// TIA Portal V17 export
// export: Created 2024-08-26T21:07:16.8648611Z, ExportSetting WithDefaults, DisplayName Totally Integrated Automation Portal, DisplayVersion V17 Update 7, DisplayName TIA Portal Openness, DisplayVersion V17 Update 7, DisplayName TIA Portal Version Control Interface, DisplayVersion V17, DisplayName SINAMICS Startdrive Advanced, DisplayVersion V17 SP2, DisplayName SINAMICS Startdrive G110M, G120, G120C, G120D, G120P, G115D, DisplayVersion V17 SP2, DisplayName SINAMICS Startdrive G130, G150, S120, S150, SINAMICS MV, S210, DisplayVersion V17 SP2, DisplayName STEP 7 Professional, DisplayVersion V17 Update 7, DisplayName STEP 7 Safety, DisplayVersion V17 Update 6, DisplayName WinCC Advanced / Unified PC, DisplayVersion V17 Update 7
FUNCTION "SCANNER CONFIG" : Void   // FC11, LAD
{ S7_Optimized_Access := 'TRUE' }
VERSION : 0.1
// stored: AutoNumber true, IsIECCheckEnabled false, SetENOAutomatically false, UDAEnableTagReadback false
   VAR_TEMP   // added for the SCL form of the ladder/FBD networks
      _w1 : Bool;
   END_VAR
BEGIN

REGION Network 1: NEST CODE READING
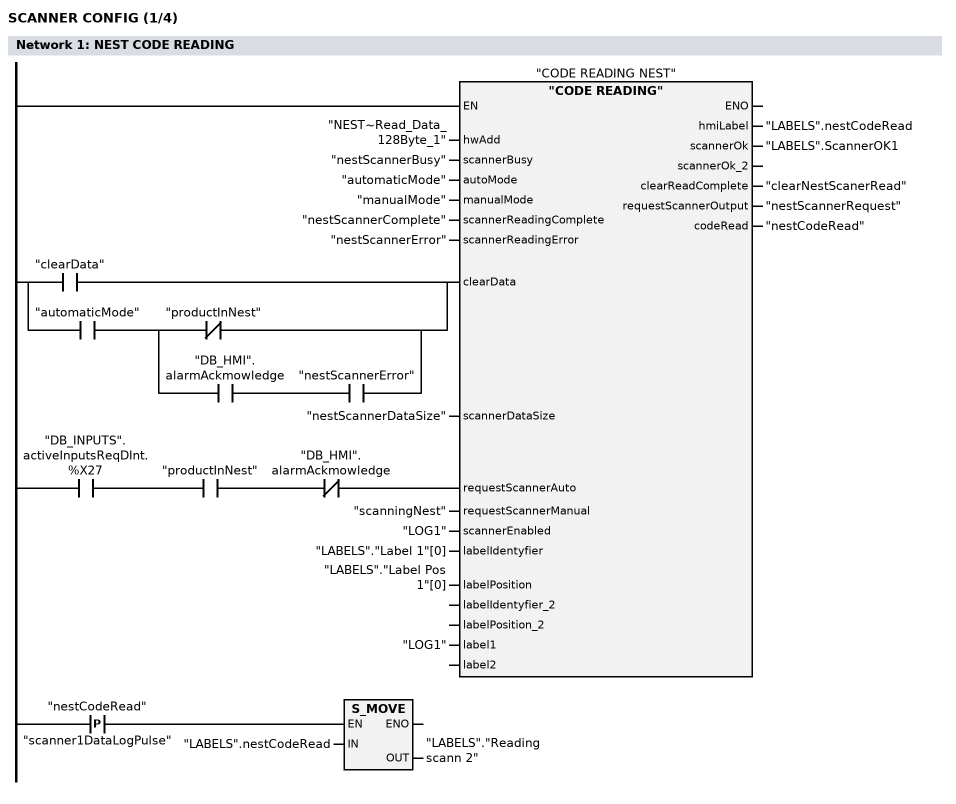
   RUNG wire#powerrail
      "CODE READING NEST"(clearData := wire#w2, requestScannerAuto := wire#w3, hwAdd := "NEST~Read_Data_128Byte_1", scannerBusy := "nestScannerBusy", autoMode := "automaticMode", manualMode := "manualMode", scannerReadingComplete := "nestScannerComplete", scannerReadingError := "nestScannerError", scannerDataSize := "nestScannerDataSize", requestScannerManual := "scanningNest", scannerEnabled := "LOG1", labelIdentyfier := "LABELS"."Label 1"[0], labelPosition := "LABELS"."Label Pos 1"[0], labelIdentyfier_2 :=, labelPosition_2 :=, label1 := "LOG1", label2 :=, hmiLabel => "LABELS".nestCodeRead, scannerOk => "LABELS".ScannerOK1, scannerOk_2 =>, clearReadComplete => "clearNestScanerRead", requestScannerOutput => "nestScannerRequest", codeRead => "nestCodeRead")
   END_RUNG
   RUNG wire#powerrail
      Contact( "clearData" )
   END_RUNG wire#w2
   RUNG wire#powerrail
      Contact( "automaticMode" )
      wire#w1
      I_Contact( "productInNest" )
   END_RUNG wire#w2
   RUNG wire#w1
      Contact( "DB_HMI".alarmAckmowledge )
      Contact( "nestScannerError" )
   END_RUNG wire#w2
   RUNG wire#powerrail
      Contact( "DB_INPUTS".activeInputsReqDInt.%X27 )
      Contact( "productInNest" )
      I_Contact( "DB_HMI".alarmAckmowledge )
   END_RUNG wire#w3
   RUNG wire#powerrail
      P_Contact(operand := "nestCodeRead", bit := "scanner1DataLogPulse")
      S_Move(in := "LABELS".nestCodeRead, out => "LABELS"."Reading scann 2")
   END_RUNG
   // the same network as SCL:
   "CODE READING NEST"(hwAdd := "NEST~Read_Data_128Byte_1",   // "CODE READING"
                       scannerBusy := "nestScannerBusy",
                       autoMode := "automaticMode",
                       manualMode := "manualMode",
                       scannerReadingComplete := "nestScannerComplete",
                       scannerReadingError := "nestScannerError",
                       clearData := "clearData" OR ("automaticMode" AND (NOT "productInNest" OR ("DB_HMI".alarmAckmowledge AND "nestScannerError"))),
                       scannerDataSize := "nestScannerDataSize",
                       requestScannerAuto := "DB_INPUTS".activeInputsReqDInt.%X27 AND "productInNest" AND NOT "DB_HMI".alarmAckmowledge,
                       requestScannerManual := "scanningNest",
                       scannerEnabled := "LOG1",
                       labelIdentyfier := "LABELS"."Label 1"[0],
                       labelPosition := "LABELS"."Label Pos 1"[0],
                       label1 := "LOG1",
                       hmiLabel => "LABELS".nestCodeRead,
                       scannerOk => "LABELS".ScannerOK1,
                       clearReadComplete => "clearNestScanerRead",
                       requestScannerOutput => "nestScannerRequest",
                       codeRead => "nestCodeRead");
   #_w1 := "nestCodeRead" AND NOT "scanner1DataLogPulse";   // rising edge of "nestCodeRead"
   "scanner1DataLogPulse" := "nestCodeRead";
   IF #_w1 THEN "LABELS"."Reading scann 2" := "LABELS".nestCodeRead; END_IF;
END_REGION

REGION Network 2: UPPER CODE READING
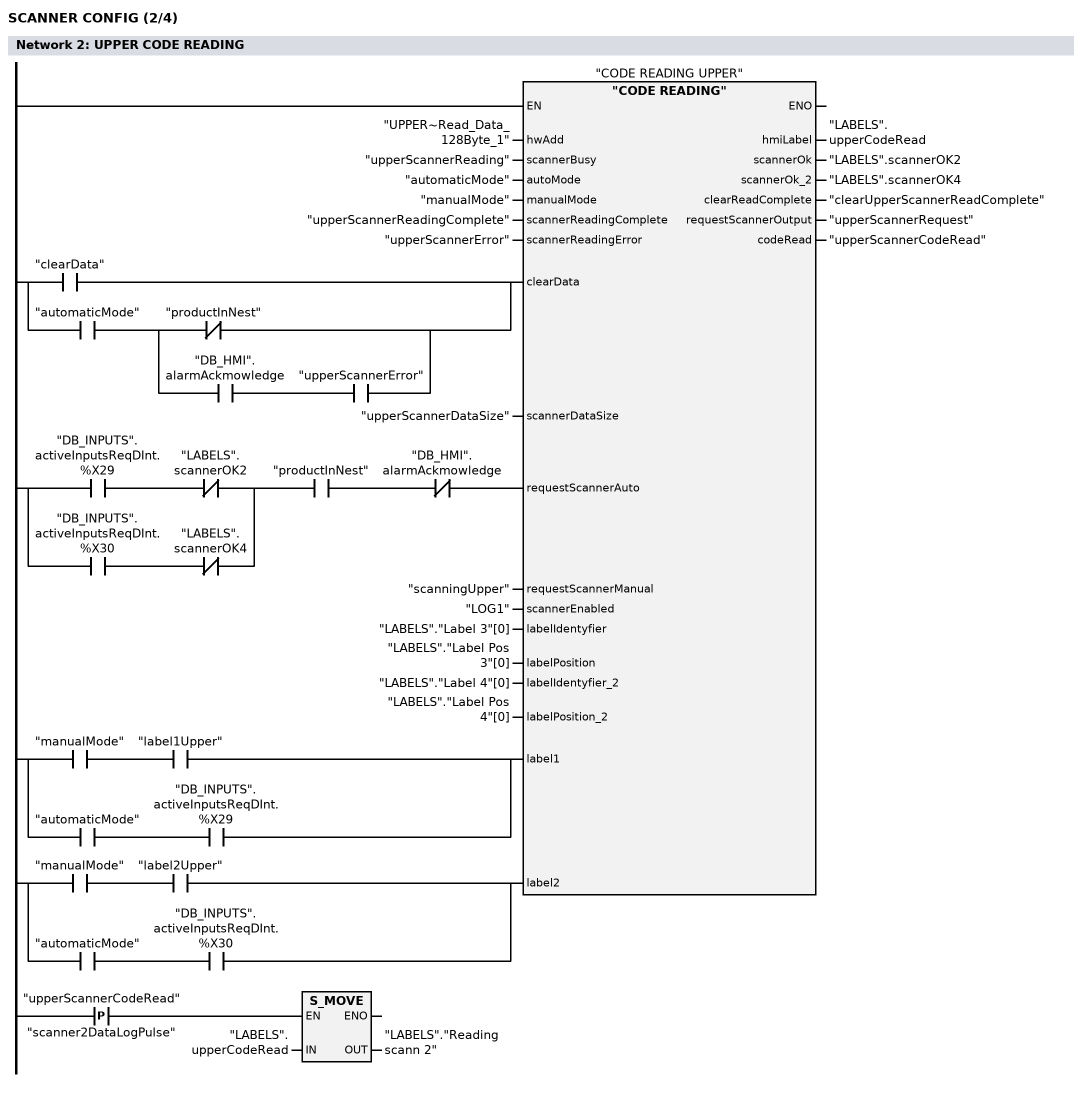
   RUNG wire#powerrail
      "CODE READING UPPER"(clearData := wire#w2, requestScannerAuto := wire#w4, label1 := wire#w5, label2 := wire#w6, hwAdd := "UPPER~Read_Data_128Byte_1", scannerBusy := "upperScannerReading", autoMode := "automaticMode", manualMode := "manualMode", scannerReadingComplete := "upperScannerReadingComplete", scannerReadingError := "upperScannerError", scannerDataSize := "upperScannerDataSize", requestScannerManual := "scanningUpper", scannerEnabled := "LOG1", labelIdentyfier := "LABELS"."Label 3"[0], labelPosition := "LABELS"."Label Pos 3"[0], labelIdentyfier_2 := "LABELS"."Label 4"[0], labelPosition_2 := "LABELS"."Label Pos 4"[0], hmiLabel => "LABELS".upperCodeRead, scannerOk => "LABELS".scannerOK2, scannerOk_2 => "LABELS".scannerOK4, clearReadComplete => "clearUpperScannerReadComplete", requestScannerOutput => "upperScannerRequest", codeRead => "upperScannerCodeRead")
   END_RUNG
   RUNG wire#powerrail
      Contact( "clearData" )
   END_RUNG wire#w2
   RUNG wire#powerrail
      Contact( "automaticMode" )
      wire#w1
      I_Contact( "productInNest" )
   END_RUNG wire#w2
   RUNG wire#w1
      Contact( "DB_HMI".alarmAckmowledge )
      Contact( "upperScannerError" )
   END_RUNG wire#w2
   RUNG wire#powerrail
      Contact( "DB_INPUTS".activeInputsReqDInt.%X29 )
      I_Contact( "LABELS".scannerOK2 )
      wire#w3
      Contact( "productInNest" )
      I_Contact( "DB_HMI".alarmAckmowledge )
   END_RUNG wire#w4
   RUNG wire#powerrail
      Contact( "DB_INPUTS".activeInputsReqDInt.%X30 )
      I_Contact( "LABELS".scannerOK4 )
   END_RUNG wire#w3
   RUNG wire#powerrail
      Contact( "manualMode" )
      Contact( "label1Upper" )
   END_RUNG wire#w5
   RUNG wire#powerrail
      Contact( "automaticMode" )
      Contact( "DB_INPUTS".activeInputsReqDInt.%X29 )
   END_RUNG wire#w5
   RUNG wire#powerrail
      Contact( "manualMode" )
      Contact( "label2Upper" )
   END_RUNG wire#w6
   RUNG wire#powerrail
      Contact( "automaticMode" )
      Contact( "DB_INPUTS".activeInputsReqDInt.%X30 )
   END_RUNG wire#w6
   RUNG wire#powerrail
      P_Contact(operand := "upperScannerCodeRead", bit := "scanner2DataLogPulse")
      S_Move(in := "LABELS".upperCodeRead, out => "LABELS"."Reading scann 2")
   END_RUNG
   // the same network as SCL:
   "CODE READING UPPER"(hwAdd := "UPPER~Read_Data_128Byte_1",   // "CODE READING"
                        scannerBusy := "upperScannerReading",
                        autoMode := "automaticMode",
                        manualMode := "manualMode",
                        scannerReadingComplete := "upperScannerReadingComplete",
                        scannerReadingError := "upperScannerError",
                        clearData := "clearData" OR ("automaticMode" AND (NOT "productInNest" OR ("DB_HMI".alarmAckmowledge AND "upperScannerError"))),
                        scannerDataSize := "upperScannerDataSize",
                        requestScannerAuto := (("DB_INPUTS".activeInputsReqDInt.%X29 AND NOT "LABELS".scannerOK2) OR ("DB_INPUTS".activeInputsReqDInt.%X30 AND NOT "LABELS".scannerOK4)) AND "productInNest" AND NOT "DB_HMI".alarmAckmowledge,
                        requestScannerManual := "scanningUpper",
                        scannerEnabled := "LOG1",
                        labelIdentyfier := "LABELS"."Label 3"[0],
                        labelPosition := "LABELS"."Label Pos 3"[0],
                        labelIdentyfier_2 := "LABELS"."Label 4"[0],
                        labelPosition_2 := "LABELS"."Label Pos 4"[0],
                        label1 := ("manualMode" AND "label1Upper") OR ("automaticMode" AND "DB_INPUTS".activeInputsReqDInt.%X29),
                        label2 := ("manualMode" AND "label2Upper") OR ("automaticMode" AND "DB_INPUTS".activeInputsReqDInt.%X30),
                        hmiLabel => "LABELS".upperCodeRead,
                        scannerOk => "LABELS".scannerOK2,
                        scannerOk_2 => "LABELS".scannerOK4,
                        clearReadComplete => "clearUpperScannerReadComplete",
                        requestScannerOutput => "upperScannerRequest",
                        codeRead => "upperScannerCodeRead");
   #_w1 := "upperScannerCodeRead" AND NOT "scanner2DataLogPulse";   // rising edge of "upperScannerCodeRead"
   "scanner2DataLogPulse" := "upperScannerCodeRead";
   IF #_w1 THEN "LABELS"."Reading scann 2" := "LABELS".upperCodeRead; END_IF;
END_REGION

REGION Network 3: ANGLE CODE READING
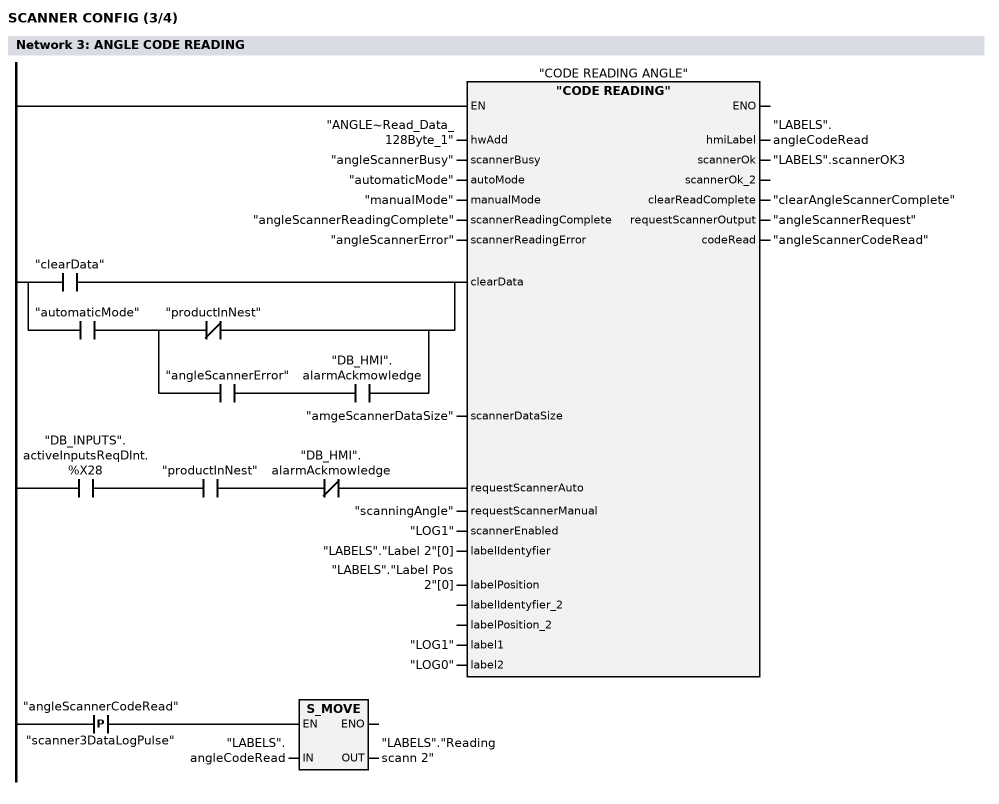
   RUNG wire#powerrail
      "CODE READING ANGLE"(clearData := wire#w2, requestScannerAuto := wire#w3, hwAdd := "ANGLE~Read_Data_128Byte_1", scannerBusy := "angleScannerBusy", autoMode := "automaticMode", manualMode := "manualMode", scannerReadingComplete := "angleScannerReadingComplete", scannerReadingError := "angleScannerError", scannerDataSize := "amgeScannerDataSize", requestScannerManual := "scanningAngle", scannerEnabled := "LOG1", labelIdentyfier := "LABELS"."Label 2"[0], labelPosition := "LABELS"."Label Pos 2"[0], labelIdentyfier_2 :=, labelPosition_2 :=, label1 := "LOG1", label2 := "LOG0", hmiLabel => "LABELS".angleCodeRead, scannerOk => "LABELS".scannerOK3, scannerOk_2 =>, clearReadComplete => "clearAngleScannerComplete", requestScannerOutput => "angleScannerRequest", codeRead => "angleScannerCodeRead")
   END_RUNG
   RUNG wire#powerrail
      Contact( "clearData" )
   END_RUNG wire#w2
   RUNG wire#powerrail
      Contact( "automaticMode" )
      wire#w1
      I_Contact( "productInNest" )
   END_RUNG wire#w2
   RUNG wire#w1
      Contact( "angleScannerError" )
      Contact( "DB_HMI".alarmAckmowledge )
   END_RUNG wire#w2
   RUNG wire#powerrail
      Contact( "DB_INPUTS".activeInputsReqDInt.%X28 )
      Contact( "productInNest" )
      I_Contact( "DB_HMI".alarmAckmowledge )
   END_RUNG wire#w3
   RUNG wire#powerrail
      P_Contact(operand := "angleScannerCodeRead", bit := "scanner3DataLogPulse")
      S_Move(in := "LABELS".angleCodeRead, out => "LABELS"."Reading scann 2")
   END_RUNG
   // the same network as SCL:
   "CODE READING ANGLE"(hwAdd := "ANGLE~Read_Data_128Byte_1",   // "CODE READING"
                        scannerBusy := "angleScannerBusy",
                        autoMode := "automaticMode",
                        manualMode := "manualMode",
                        scannerReadingComplete := "angleScannerReadingComplete",
                        scannerReadingError := "angleScannerError",
                        clearData := "clearData" OR ("automaticMode" AND (NOT "productInNest" OR ("angleScannerError" AND "DB_HMI".alarmAckmowledge))),
                        scannerDataSize := "amgeScannerDataSize",
                        requestScannerAuto := "DB_INPUTS".activeInputsReqDInt.%X28 AND "productInNest" AND NOT "DB_HMI".alarmAckmowledge,
                        requestScannerManual := "scanningAngle",
                        scannerEnabled := "LOG1",
                        labelIdentyfier := "LABELS"."Label 2"[0],
                        labelPosition := "LABELS"."Label Pos 2"[0],
                        label1 := "LOG1",
                        label2 := "LOG0",
                        hmiLabel => "LABELS".angleCodeRead,
                        scannerOk => "LABELS".scannerOK3,
                        clearReadComplete => "clearAngleScannerComplete",
                        requestScannerOutput => "angleScannerRequest",
                        codeRead => "angleScannerCodeRead");
   #_w1 := "angleScannerCodeRead" AND NOT "scanner3DataLogPulse";   // rising edge of "angleScannerCodeRead"
   "scanner3DataLogPulse" := "angleScannerCodeRead";
   IF #_w1 THEN "LABELS"."Reading scann 2" := "LABELS".angleCodeRead; END_IF;
END_REGION

REGION Network 4: Move values to HMI
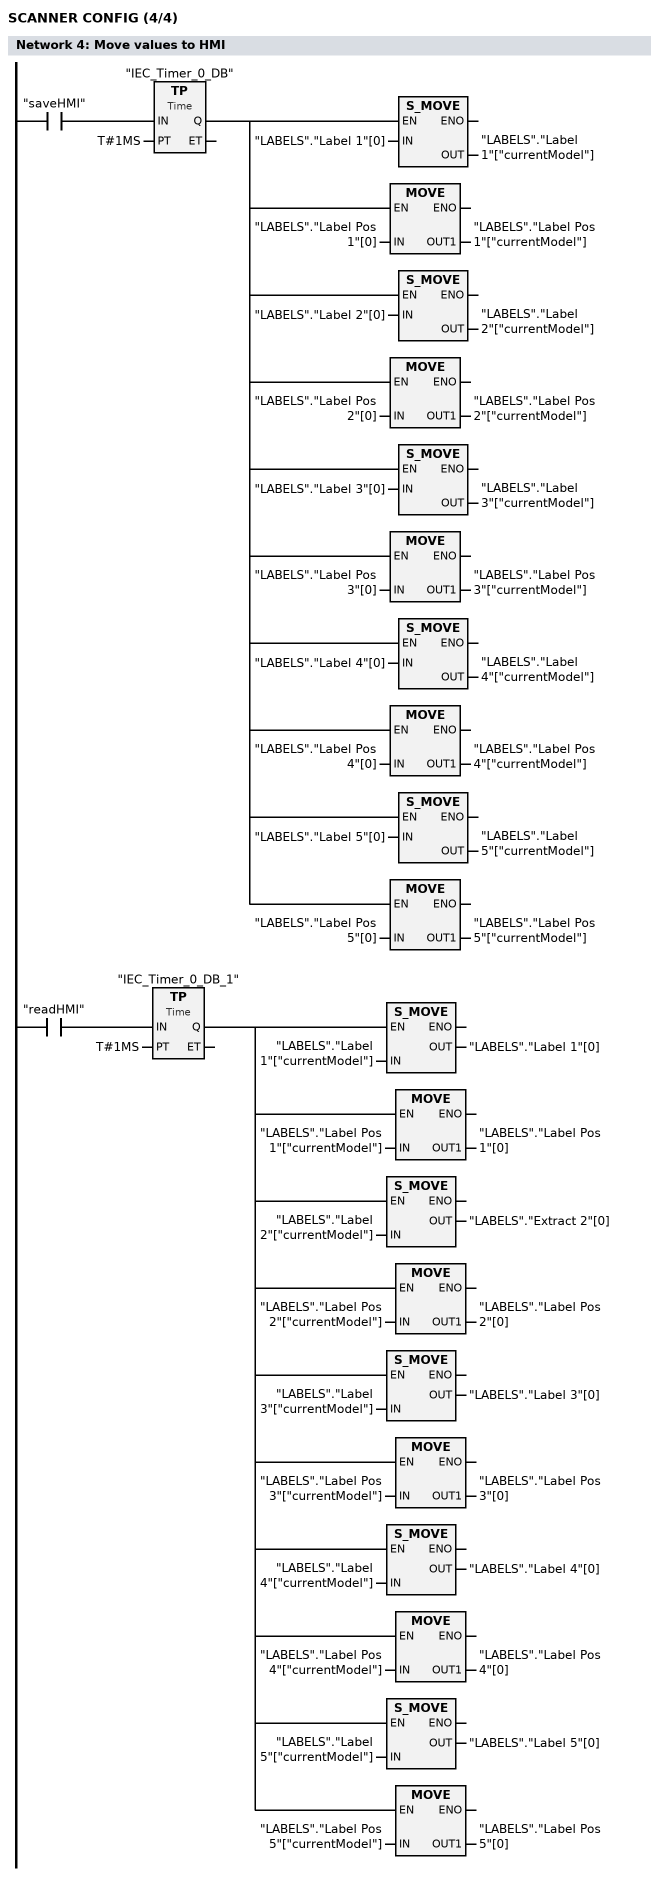
   RUNG wire#powerrail
      Contact( "saveHMI" )
      { S7_Templates := "time_type := Time" } "IEC_Timer_0_DB".TP(pt := T#1MS, et =>)
      wire#w1
      S_Move(in := "LABELS"."Label 1"[0], out => "LABELS"."Label 1"["currentModel"])
   END_RUNG
   RUNG wire#w1
      Move(in := "LABELS"."Label Pos 1"[0], out1 => "LABELS"."Label Pos 1"["currentModel"])
   END_RUNG
   RUNG wire#w1
      S_Move(in := "LABELS"."Label 2"[0], out => "LABELS"."Label 2"["currentModel"])
   END_RUNG
   RUNG wire#w1
      Move(in := "LABELS"."Label Pos 2"[0], out1 => "LABELS"."Label Pos 2"["currentModel"])
   END_RUNG
   RUNG wire#w1
      S_Move(in := "LABELS"."Label 3"[0], out => "LABELS"."Label 3"["currentModel"])
   END_RUNG
   RUNG wire#w1
      Move(in := "LABELS"."Label Pos 3"[0], out1 => "LABELS"."Label Pos 3"["currentModel"])
   END_RUNG
   RUNG wire#w1
      S_Move(in := "LABELS"."Label 4"[0], out => "LABELS"."Label 4"["currentModel"])
   END_RUNG
   RUNG wire#w1
      Move(in := "LABELS"."Label Pos 4"[0], out1 => "LABELS"."Label Pos 4"["currentModel"])
   END_RUNG
   RUNG wire#w1
      S_Move(in := "LABELS"."Label 5"[0], out => "LABELS"."Label 5"["currentModel"])
   END_RUNG
   RUNG wire#w1
      Move(in := "LABELS"."Label Pos 5"[0], out1 => "LABELS"."Label Pos 5"["currentModel"])
   END_RUNG
   RUNG wire#powerrail
      Contact( "readHMI" )
      { S7_Templates := "time_type := Time" } "IEC_Timer_0_DB_1".TP(pt := T#1MS, et =>)
      wire#w2
      S_Move(in := "LABELS"."Label 1"["currentModel"], out => "LABELS"."Label 1"[0])
   END_RUNG
   RUNG wire#w2
      Move(in := "LABELS"."Label Pos 1"["currentModel"], out1 => "LABELS"."Label Pos 1"[0])
   END_RUNG
   RUNG wire#w2
      S_Move(in := "LABELS"."Label 2"["currentModel"], out => "LABELS"."Extract 2"[0])
   END_RUNG
   RUNG wire#w2
      Move(in := "LABELS"."Label Pos 2"["currentModel"], out1 => "LABELS"."Label Pos 2"[0])
   END_RUNG
   RUNG wire#w2
      S_Move(in := "LABELS"."Label 3"["currentModel"], out => "LABELS"."Label 3"[0])
   END_RUNG
   RUNG wire#w2
      Move(in := "LABELS"."Label Pos 3"["currentModel"], out1 => "LABELS"."Label Pos 3"[0])
   END_RUNG
   RUNG wire#w2
      S_Move(in := "LABELS"."Label 4"["currentModel"], out => "LABELS"."Label 4"[0])
   END_RUNG
   RUNG wire#w2
      Move(in := "LABELS"."Label Pos 4"["currentModel"], out1 => "LABELS"."Label Pos 4"[0])
   END_RUNG
   RUNG wire#w2
      S_Move(in := "LABELS"."Label 5"["currentModel"], out => "LABELS"."Label 5"[0])
   END_RUNG
   RUNG wire#w2
      Move(in := "LABELS"."Label Pos 5"["currentModel"], out1 => "LABELS"."Label Pos 5"[0])
   END_RUNG
   // the same network as SCL:
   "IEC_Timer_0_DB".TP(IN := "saveHMI", PT := T#1MS);
   IF "IEC_Timer_0_DB".Q THEN
       "LABELS"."Label 1"["currentModel"] := "LABELS"."Label 1"[0];
       "LABELS"."Label Pos 1"["currentModel"] := "LABELS"."Label Pos 1"[0];
       "LABELS"."Label 2"["currentModel"] := "LABELS"."Label 2"[0];
       "LABELS"."Label Pos 2"["currentModel"] := "LABELS"."Label Pos 2"[0];
       "LABELS"."Label 3"["currentModel"] := "LABELS"."Label 3"[0];
       "LABELS"."Label Pos 3"["currentModel"] := "LABELS"."Label Pos 3"[0];
       "LABELS"."Label 4"["currentModel"] := "LABELS"."Label 4"[0];
       "LABELS"."Label Pos 4"["currentModel"] := "LABELS"."Label Pos 4"[0];
       "LABELS"."Label 5"["currentModel"] := "LABELS"."Label 5"[0];
       "LABELS"."Label Pos 5"["currentModel"] := "LABELS"."Label Pos 5"[0];
   END_IF;
   "IEC_Timer_0_DB_1".TP(IN := "readHMI", PT := T#1MS);
   IF "IEC_Timer_0_DB_1".Q THEN
       "LABELS"."Label 1"[0] := "LABELS"."Label 1"["currentModel"];
       "LABELS"."Label Pos 1"[0] := "LABELS"."Label Pos 1"["currentModel"];
       "LABELS"."Extract 2"[0] := "LABELS"."Label 2"["currentModel"];
       "LABELS"."Label Pos 2"[0] := "LABELS"."Label Pos 2"["currentModel"];
       "LABELS"."Label 3"[0] := "LABELS"."Label 3"["currentModel"];
       "LABELS"."Label Pos 3"[0] := "LABELS"."Label Pos 3"["currentModel"];
       "LABELS"."Label 4"[0] := "LABELS"."Label 4"["currentModel"];
       "LABELS"."Label Pos 4"[0] := "LABELS"."Label Pos 4"["currentModel"];
       "LABELS"."Label 5"[0] := "LABELS"."Label 5"["currentModel"];
       "LABELS"."Label Pos 5"[0] := "LABELS"."Label Pos 5"["currentModel"];
   END_IF;
END_REGION
END_FUNCTION
